{attribute 'Tc2GvlVarNames'}
VAR_GLOBAL
	CheckBounds_ErrCnt 			: DINT;
	CheckByteZeroDiv_ErrCnt 		: DINT;
	CheckDWordZeroDiv_ErrCnt 	: DINT;
	CheckRealZeroDiv_ErrCnt 		: DINT;
	CheckWordZeroDiv_ErrCnt 		: DINT;
	CheckRangeSigned_ErrCnt		: DINT;
	CheckRangeUnsigned_ErrCnt	: DINT;
END_VAR

(* stored: Version 1.1.0.1, ProductVersion 3.1.4024.15
   GVL Global_Checks: Id {cc1c4075-d9f2-48f1-b254-55f90b7bf63a} *)
